{attribute 'qualified_only'}
VAR_GLOBAL
//E-StopAlarm 장비 정지
	E_STOP_Alarm01			: BOOL	;		//EMO-Switch ON
	E_STOP_Alarm02			: BOOL	;		//Door Open
	E_STOP_Alarm03			: BOOL	;	
	E_STOP_Alarm04			: BOOL	;
	E_STOP_Alarm05			: BOOL	;
	E_STOP_Alarm06			: BOOL	;	
	E_STOP_Alarm07			: BOOL	;
	E_STOP_Alarm08			: BOOL	;
	E_STOP_Alarm09			: BOOL	;
	E_STOP_Alarm10			: BOOL	;		//Vision 통신 이상
	E_STOP_Alarm11			: BOOL	;
	E_STOP_Alarm12			: BOOL	;
	E_STOP_Alarm13			: BOOL	;
	E_STOP_Alarm14			: BOOL	;
	E_STOP_Alarm15			: BOOL	;
//Display Alarm 알람
	Display_Alarm01			: BOOL	;		
	Display_Alarm02			: BOOL	;
	Display_Alarm03			: BOOL	;
	Display_Alarm04			: BOOL	;
	Display_Alarm05			: BOOL	;
	Display_Alarm06			: BOOL	;
	Display_Alarm07			: BOOL	;
	Display_Alarm08			: BOOL	;
	Display_Alarm09			: BOOL	;
	Display_Alarm10			: BOOL	;		//Vision 측정 NG
	Display_Alarm11			: BOOL	;
	Display_Alarm12			: BOOL	;
	Display_Alarm13			: BOOL	;
	Display_Alarm14			: BOOL	;	
	Display_Alarm15			: BOOL	;
//Axis01 Motor Alarm
	Axis01_Total_Alarm		: BOOL	;		
	Axis01_Alarm01			: BOOL	;		
	Axis01_Alarm02			: BOOL	;
	Axis01_Alarm03			: BOOL	;		
	Axis01_Alarm04			: BOOL	;		
	Axis01_Alarm05			: BOOL	;		
	Axis01_Alarm06			: BOOL	;		
	Axis01_Alarm07			: BOOL	;		
	Axis01_Alarm08			: BOOL	;		
	Axis01_Alarm09			: BOOL	;		
	Axis01_Alarm10			: BOOL	;		
//Axis02 Motor Alarm
	Axis02_Total_Alarm		: BOOL	;		
	Axis02_Alarm01			: BOOL	;		
	Axis02_Alarm02			: BOOL	;
	Axis02_Alarm03			: BOOL	;		
	Axis02_Alarm04			: BOOL	;		
	Axis02_Alarm05			: BOOL	;		
	Axis02_Alarm06			: BOOL	;		
	Axis02_Alarm07			: BOOL	;		
	Axis02_Alarm08			: BOOL	;		
	Axis02_Alarm09			: BOOL	;		
	Axis02_Alarm10			: BOOL	;		
//Axis03 Motor Alarm
	Axis03_Total_Alarm		: BOOL	;		
	Axis03_Alarm01			: BOOL	;		
	Axis03_Alarm02			: BOOL	;
	Axis03_Alarm03			: BOOL	;		
	Axis03_Alarm04			: BOOL	;		
	Axis03_Alarm05			: BOOL	;		
	Axis03_Alarm06			: BOOL	;		
	Axis03_Alarm07			: BOOL	;		
	Axis03_Alarm08			: BOOL	;		
	Axis03_Alarm09			: BOOL	;		
	Axis03_Alarm10			: BOOL	;		
//Axis04 Motor Alarm
	Axis04_Total_Alarm		: BOOL	;		
	Axis04_Alarm01			: BOOL	;		
	Axis04_Alarm02			: BOOL	;
	Axis04_Alarm03			: BOOL	;		
	Axis04_Alarm04			: BOOL	;		
	Axis04_Alarm05			: BOOL	;		
	Axis04_Alarm06			: BOOL	;		
	Axis04_Alarm07			: BOOL	;		
	Axis04_Alarm08			: BOOL	;		
	Axis04_Alarm09			: BOOL	;		
	Axis04_Alarm10			: BOOL	;		
//Axis05 Motor Alarm
	Axis05_Total_Alarm		: BOOL	;		
	Axis05_Alarm01			: BOOL	;		
	Axis05_Alarm02			: BOOL	;
	Axis05_Alarm03			: BOOL	;		
	Axis05_Alarm04			: BOOL	;		
	Axis05_Alarm05			: BOOL	;		
	Axis05_Alarm06			: BOOL	;		
	Axis05_Alarm07			: BOOL	;		
	Axis05_Alarm08			: BOOL	;		
	Axis05_Alarm09			: BOOL	;		
	Axis05_Alarm10			: BOOL	;		
	E_STOP_Total_Alarm		: BOOL	;
	EMO_SWitch				: BOOL	;
END_VAR

(* stored: Version 1.1.0.1, ProductVersion 3.1.4024.15
   GVL GVL_Alarm_1: Id {eba1c83d-5da1-4916-bb8e-4b625d3c6815} *)
